// TwinCAT 3 PLC project pruebaAlmacenje
// ProgramVersion: 3.1.4024.0
// libraries:
//   Tc2_Standard, * (Beckhoff Automation GmbH)
//   Tc2_System, * (Beckhoff Automation GmbH)
//   Tc3_Module, * (Beckhoff Automation GmbH)
//   VisuSymbols,3.5.10.0,System
// project tree:
//   / GlobalTextList.TcGTLO, PlcTask.TcTTO (not stored), Visualization Manager.TcVMO (not stored)
//   GVLs/ GVLvar.TcGVL
//   POUs/ inicializarPosOcupEstanteria.TcPOU, MAIN.TcPOU, posicionEstanteria.TcPOU, distanciaBaldas.TcPOU
//   VISUs/ equivalenciaBaldaOcupada.TcTLO, HMI.TcVIS
// real-time tasks:
//   TASK PlcTask: cycle T#10ms, priority 20, ADS port 350

// ---- GVLs/GVLvar.TcGVL
{attribute 'qualified_only'}
VAR_GLOBAL
	
	// Cuadro
	{attribute 'OPC.UA.DA' := '1'}
	botonStart : BOOL;
	{attribute 'OPC.UA.DA' := '1'}
	botonStop : BOOL;
	{attribute 'OPC.UA.DA' := '1'}
	botonReset : BOOL; 
	{attribute 'OPC.UA.DA' := '1'}
	seta: BOOL;
	{attribute 'OPC.UA.DA' := '1'}
	luzVerde : BOOL;
	{attribute 'OPC.UA.DA' := '1'}
	luzAmarillo : BOOL;
	{attribute 'OPC.UA.DA' := '1'}
	luzRoja : BOOL;
	{attribute 'OPC.UA.DA' := '1'}
	luzBotonStart : BOOL;
	{attribute 'OPC.UA.DA' := '1'}
	luzBotonStop :  BOOL;
	{attribute 'OPC.UA.DA' := '1'}
	luzBotonReset : BOOL;
	{attribute 'OPC.UA.DA' := '1'}
	modoManual : BOOL;
	{attribute 'OPC.UA.DA' := '1'}
	modoAuto : BOOL;
	
	

	// Estanterias
	estanteria: ARRAY[1..6,1..6] OF ARRAY[1..2] OF REAL;
	baldasOcupadas : ARRAY [1..6,1..3] OF BOOL;
	
	// Cintas
	{attribute 'OPC.UA.DA' := '1'}
	cinta : BOOL;
	{attribute 'OPC.UA.DA' := '1'}
	cintaTransportadoraPalet : BOOL; 

	// Grua
	{attribute 'OPC.UA.DA' := '1'}
	moveForksLeft : BOOL; // horquilla hacia ixquierda
	{attribute 'OPC.UA.DA' := '1'}
	moveForksRight : BOOL; // hoquilla hacia derecha
	//{attribute 'OPC.UA.DA' := '1'}
	//elevacionLigeraPlataforma : BOOL;
	{attribute 'OPC.UA.DA' := '1'}
	movingZ : REAL; // actual poscion en Z
	{attribute 'OPC.UA.DA' := '1'}
	movingX : REAL; // actual posicion en X
	{attribute 'OPC.UA.DA' := '1'}
	forkLeftLimit : BOOL; 
	{attribute 'OPC.UA.DA' := '1'}
	forkMiddleLimit : BOOL;
	{attribute 'OPC.UA.DA' := '1'}
	forkRightLimit : BOOL;
	{attribute 'OPC.UA.DA' := '1'}
	setPointX : REAL; // movimientp columnas (horizontal)
	{attribute 'OPC.UA.DA' := '1'}
	setPointZ : REAL; // movimeinto filas (vertical)
	
	//sensores
	{attribute 'OPC.UA.DA' := '1'}
	sensorEntradaGrua : bool;


END_VAR

// ---- POUs/inicializarPosOcupEstanteria.TcPOU
FUNCTION_BLOCK inicializarPosOcupEstanteria
VAR_INPUT
END_VAR
VAR_OUTPUT
END_VAR
VAR
	i: INT;
	fila: INT;
	col: INT;
END_VAR

// Se inicializan las posicones del amlmcen a false
// por defecto se empieza con el almacen vacio
FOR fila := 1 TO 6 DO
    FOR col := 1 TO 3 DO
        // la primera posicion libre 
		 GVLvar.baldasOcupadas[fila,col] := FALSE;
    END_FOR
END_FOR

END_FUNCTION_BLOCK

// ---- POUs/MAIN.TcPOU
PROGRAM MAIN
VAR
	enclaveStart: BOOL;
	timerColumna: TON;
	posicionEst : ARRAY[1..4] OF REAL;
	distBaldas : distanciaBaldas();
	iniPosOcupEst : inicializarPosOcupEstanteria();
	cargando: BOOL;
	flancoMovingX : F_TRIG;
	flancoMovingZ : F_TRIG;
	movingZ: BOOL;
	movingX: BOOL;
	descragandoElem: BOOL;
	descargandoElem: BOOL;
	elemDescargado: BOOL;
	state: INT := 1;
	posInicialZ : real := 0.2;
	horquillaExtendida: BOOL;
	timerExternsionHorquilla: TON;
	startTimerHorquilla: BOOL;
	timerExtension: BOOL;
	posActual: REAL;
	bajarHorquilla: BOOL;
	timerBajarHorquilla: TON;
	incfementoBaizadaH : REAL := 0.4;
	enPosicoin: BOOL;
	posmovingZ: REAL;
	luzStart :bool;
	luzReset: BOOL;
	luzStop : bool;
	luzVerde: BOOL;
	luzAmarilla: BOOL;
	luzRoja: BOOL;
	emergencia: BOOL;
	cinta:bool;
	setPointX: REAL;
	setPointZ: REAL;
	cintaTransportadoraPalet: BOOL;
	botonReset: BOOL;
	seta : bool;
	botonStart: BOOL;
	botonStop: BOOL;
	filaEstanteria: INT;
	colEstanteria: INT;
	moving: REAL;
END_VAR

VAR PERSISTENT
	elemCargado: BOOL;
END_VAR

// ----------------------------- Logica Botones ----------------------------------------

//Luces Botons
luzStart := FALSE;
luzStop := FALSE;
luzReset:=FALSE;

(*Boton start 



*)
IF GVLvar.botonStart AND NOT emergencia THEN
	luzStart:= TRUE;
	luzVerde := TRUE;
	luzAmarilla := FALSE;
	luzRoja := FALSE;
	enclaveStart := TRUE;
	cinta := TRUE;
	cintaTransportadoraPalet := TRUE; 
	distBaldas();
	iniPosOcupEst();
	setPointZ := 0.2;
END_IF

IF NOT GVLvar.botonStop AND NOT emergencia THEN
	luzStop := TRUE;
	luzVerde := FALSE;
	luzAmarilla := TRUE;
	luzRoja := FALSE;
	enclaveStart := FALSE;
	cinta := FALSE;
	cintaTransportadoraPalet := FALSE;
END_IF


IF  NOT GVLvar.seta THEN
	luzRoja:= TRUE;
	luzVerde := FALSE;
	luzAmarilla := FALSE;
	
	emergencia := TRUE;
	cinta := FALSE;
	cintaTransportadoraPalet := FALSE	; 
	enclaveStart := FALSE;
END_IF


IF  GVLvar.seta AND emergencia THEN
	IF GVLvar.botonReset THEN
		emergencia := FALSE;
		cinta := TRUE;
		cintaTransportadoraPalet := TRUE; 
		enclaveStart := TRUE;
		luzRoja := FALSE;
		luzVerde := TRUE;
		luzAmarilla := FALSE;
	END_IF	
END_IF

// ---------------------------------------------------------------------

IF enclaveStart THEN
	

	CASE state OF
	
		// 1. Esperando Start
		1: 
//			IF GVLvar.botonStart THEN
//				enclaveStart := TRUE;
//				GVLvar.cinta := TRUE;
//				distBaldas();
//				iniPosOcupEst();
//				GVLvar.setPointZ := 0.3;
//				state := 2;  // pasar al siguiente estado
//			END_IF
			setPointZ := posInicialZ;
			state := 2;  // pasar al siguiente estado
			
		// 2. Espera caja en la entrada
		2:
			IF GVLvar.sensorEntradaGrua THEN
				cinta := FALSE;
				cintaTransportadoraPalet := FALSE;
				GVLvar.moveForksRight := TRUE;
				state := 3;
			END_IF
	
		// 3. Horquilla desplegando
		3:
			IF GVLvar.forkRightLimit THEN
				setPointZ := posInicialZ + 0.2;
				startTimerHorquilla := TRUE;
			END_IF
			
			timerExternsionHorquilla (IN:=startTimerHorquilla, PT:= T#2S);
			
			horquillaExtendida :=  (GVLvar.movingZ = (posInicialZ + 0.2)) OR (GVLvar.movingZ > ((posInicialZ + 0.2)-0.05)) OR (GVLvar.movingZ < ((posInicialZ + 0.2)+0.05));
			//IF GVLvar.movingZ = (posInicialZ + 0.2) THEN
			IF timerExternsionHorquilla.Q AND horquillaExtendida THEN
				GVLvar.moveForksRight := FALSE;
				elemCargado := TRUE;
				startTimerHorquilla := FALSE;
				state := 4;
			END_IF
			
//			IF GVLvar.forkMiddleLimit  AND elemCargado THEN 
				
				
//			END_IF
	
		// 4. Calcular posición libre y mover X/Z
		4:
			IF elemCargado AND GVLvar.forkMiddleLimit THEN 
				posicionEst := posicionEstanteria();
				// Si devuelve una posicion valida
				IF posicionEst[1]<>0 AND posicionEst[2]<>0 THEN
					setPointX := posicionEst[1];   // columna (X)
					setPointZ := posicionEst[2]+0.4;   // fila (Z)
					filaEstanteria := TO_INT(posicionEst[3]);
					colEstanteria := TO_INT(posicionEst[4]);
					elemCargado := FALSE;
					descargandoElem := TRUE;
					state := 5;
				END_IF
			END_IF
	
		// 5. Esperar llegar a destino
		5:
			 movingX := (GVLvar.movingX = posicionEst[1]) OR (GVLvar.movingX > (posicionEst[1]-0.05) AND GVLvar.movingX < posicionEst[1]) OR (GVLvar.movingX < (posicionEst[1]+0.05)AND GVLvar.movingX > posicionEst[1]) ;
			 movingZ := (GVLvar.movingZ = posicionEst[2]+0.4) OR (GVLvar.movingZ > (posicionEst[2]-0.05+0.4) AND GVLvar.movingZ < posicionEst[2]+0.4) OR (GVLvar.movingZ < (posicionEst[2]+0.05+0.4) AND GVLvar.movingZ > posicionEst[2]+0.4);
			 
			 
			IF movingZ AND movingX AND descargandoElem THEN
				GVLvar.moveForksLeft := TRUE;
				bajarHorquilla := TRUE;
				state := 6;
			END_IF
			
			
		6:	
			//timerBajarHorquilla (IN:= bajarHorquilla, PT:=T#2S);
			
			//IF  enPosicoin AND GVLvar.forkMiddleLimit THEN  
			IF GVLvar.forkLeftLimit THEN
				 moving := GVLvar.movingZ;
				IF moving > 0 THEN 
					setPointZ := GVLvar.movingZ - incfementoBaizadaH ;	
				END_IF
				descargandoElem := FALSE;
				bajarHorquilla := FALSE;
				state := 7;
			END_IF
			
		// 6. Horquilla descargando
		7:
			posmovingZ := GVLvar.movingZ;	
			enPosicoin  := (posmovingZ = posicionEst[2]) OR (posmovingZ > (posicionEst[2] -0.05) AND posmovingZ < posicionEst[2]) OR (posmovingZ < (posicionEst[2]+0.05) AND posmovingZ > posicionEst[2]);
			 
			IF GVLvar.forkLeftLimit AND enPosicoin THEN
				GVLvar.moveForksLeft := FALSE;
				elemDescargado := TRUE;
				state := 8;
       		END_IF
			
		
			
		// 7. Volver a origen
		8:
			IF elemDescargado AND GVLvar.forkMiddleLimit THEN
				setPointX := 0.0;
				setPointZ :=posInicialZ;
				elemDescargado := FALSE;
				cinta := TRUE;
				cintaTransportadoraPalet := TRUE; 
				state := 2;
			END_IF
	
	//    // 8. Reanudar cinta y volver a esperar
	//    8:
	//        IF (GVLvar.movingX = 0.0) AND (GVLvar.movingZ = 0.3) THEN
	//            GVLvar.cinta := TRUE;
	//            state := 2;   // vuelve a esperar siguiente caja
	//        END_IF
	
		// Estado por defecto (seguridad)
		ELSE
			state := 1;
	
	END_CASE
END_IF


// ----------------------------- Actualizar Salidas  ----------------------------------------
GVLvar.setPointX := setPointX;
GVLvar.setPointZ := setPointZ;

GVLvar.luzAmarillo := luzAmarilla;
GVLvar.luzVerde := luzVerde;
GVLvar.luzRoja := luzRoja;
GVLvar.luzBotonReset := luzReset;
GVLvar.luzBotonStart := luzStart;
GVLvar.luzBotonStop := luzStop;

GVLvar.cinta := cinta;
GVLvar.cintaTransportadoraPalet := cintaTransportadoraPalet;


//GVLvar.seta := seta;
//GVLvar.botonReset := botonReset;
//GVLvar.botonStart := botonStart;
//GVLvar.botonStop := botonStop:

END_PROGRAM

// ---- POUs/distanciaBaldas.TcPOU
FUNCTION_BLOCK distanciaBaldas
VAR_INPUT
END_VAR
VAR_OUTPUT
END_VAR
VAR
END_VAR

// Fila 1
GVLvar.estanteria[1,1][1] := 1.55;  GVLvar.estanteria[1,1][2] := 0.5;
GVLvar.estanteria[1,2][1] := 2.6;  GVLvar.estanteria[1,2][2] := 0.5;
GVLvar.estanteria[1,3][1] := 3.7;  GVLvar.estanteria[1,3][2] := 0.5;

// Fila 2
GVLvar.estanteria[2,1][1] := 1.55;  GVLvar.estanteria[2,1][2] := 2.1;
GVLvar.estanteria[2,2][1] := 2.6;  GVLvar.estanteria[2,2][2] := 2.1;
GVLvar.estanteria[2,3][1] := 3.7;  GVLvar.estanteria[2,3][2] := 2.1;

// Fila 3
GVLvar.estanteria[3,1][1] := 1.65;  GVLvar.estanteria[3,1][2] := 3.9;
GVLvar.estanteria[3,2][1] := 2.6;  GVLvar.estanteria[3,2][2] := 3.9;
GVLvar.estanteria[3,3][1] := 3.7;  GVLvar.estanteria[3,3][2] := 3.9;

// Fila 4
GVLvar.estanteria[4,1][1] := 1.6;  GVLvar.estanteria[4,1][2] := 5.6;
GVLvar.estanteria[4,2][1] := 2.6;  GVLvar.estanteria[4,2][2] := 5.6;
GVLvar.estanteria[4,3][1] := 3.7;  GVLvar.estanteria[4,3][2] := 5.6;

// Fila 5
GVLvar.estanteria[5,1][1] := 1.6;  GVLvar.estanteria[5,1][2] := 8.3;
GVLvar.estanteria[5,2][1] := 2.6;  GVLvar.estanteria[5,2][2] := 8.3;
GVLvar.estanteria[5,3][1] := 3.7;  GVLvar.estanteria[5,3][2] := 8.3;

// Fila 6
GVLvar.estanteria[6,1][1] := 1.6;  GVLvar.estanteria[6,1][2] := 8.7;
GVLvar.estanteria[6,2][1] := 2.6;  GVLvar.estanteria[6,2][2] := 8.7;
GVLvar.estanteria[6,3][1] := 3.7;  GVLvar.estanteria[6,3][2] := 8.7;

END_FUNCTION_BLOCK

// ---- POUs/posicionEstanteria.TcPOU
FUNCTION posicionEstanteria : Array[1..4] of real
VAR_INPUT
END_VAR
VAR
	posicion : ARRAY[1..2] OF REAL;
	// 1 - posicion en X (horizontal)
	// 2 - posicoin en Z (vertical)
	fila: DINT;
	arr2D: INT;
	col: DINT;
	encontrado: BOOL;
END_VAR

encontrado  := FALSE;
FOR fila := 1 TO 6 DO
    FOR col := 1 TO 3 DO
        // la primera posicion libre 
		IF GVLvar.baldasOcupadas[fila,col] = FALSE  AND encontrado = FALSE THEN
			posicionEstanteria[1] := GVLvar.estanteria[fila,col][1];
			posicionEstanteria[2] := GVLvar.estanteria[fila,col][2];
			posicionEstanteria[3] := TO_REAL(fila) ;
			posicionEstanteria[4] := TO_REAL(col);
			
			GVLvar.baldasOcupadas[fila,col] := TRUE;
			encontrado := TRUE;
			EXIT;
//		ELSE 
//			posicionEstanteria := [0,0];
		END_IF
    END_FOR
END_FOR

END_FUNCTION

// ---- GlobalTextList.TcGTLO
TEXTLIST GlobalTextList
  538 = '%B'
  557 = '%b'
  838 = '%i'
  837 = 'Cargando Palet'
  351 = 'Descargando Palet'
  912 = 'ESTANTERÍA'
  378 = 'FiColumnala'
  976 = 'Fila'
  655 = 'GRÚA'
  699 = 'GRÚA DESPLAZANDOSE A'
  528 = 'Horquilla en reposo'
  343 = 'Horquilla extendida Dcha'
  803 = 'Horquilla extendida Izq'
  777 = 'Indicador de mesa giratoria orientada a 90º'
  953 = 'Indicador de mesa giratoria orinetada a 0ª (posicion de reposo)'
  894 = 'Indicador de un palet sobre la mesa giratoria'
  359 = 'Mesa en 0º'
  512 = 'Mesa en 90º'
  134 = 'MESA GIRATORIA'
  194 = 'Palet en Mesa'
  465 = 'Posicion'
  379 = 'Posición '
  139 = 'Reset'
  163 = 'Seta'
  56 = 'Seta Emergencia'
  759 = 'Start'
  420 = 'Stop'
END_TEXTLIST

// ---- VISUs/equivalenciaBaldaOcupada.TcTLO
TEXTLIST equivalenciaBaldaOcupada
  TRUE = 'Ocupada'
  FALSE = 'Libre'
   = ''
END_TEXTLIST

// ---- VISUs/HMI.TcVIS
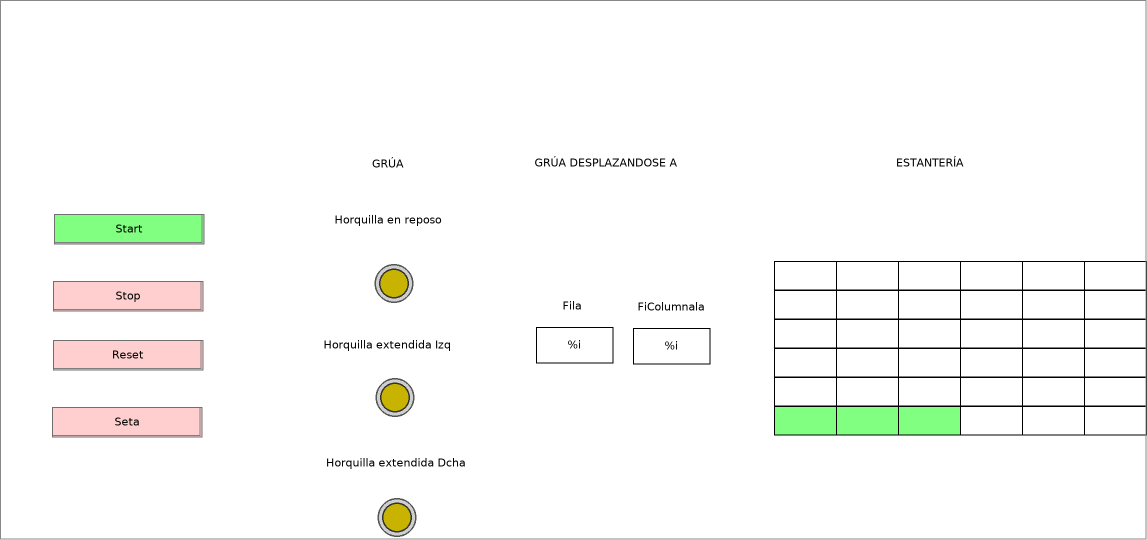
VISUALIZATION HMI  // 1147x540
    Button (54,214 150x30), "Start"
        toggle GVLvar.botonStart
    Button (53,281 150x30), "Stop", colour toggle: NOT GVLvars.botonStop
        toggle GVLvar.botonStop
    Button (53,340 150x30), "Reset", colour toggle: GVLvars.botonReset
        toggle GVLvar.botonReset
    Button (52,407 150x30), "Seta", colour toggle: GVLvars.seta
        toggle not GVLvars.seta
    Lamp1 (368,261 52x45), tooltip "Indicador de un palet sobre la mesa giratoria", variable: GVLvars.frontLimit, style: Lamp-Lamp1-Yellow
    Label (313,149 150x30), "GRÚA"
    Lamp1 (369,375 52x45), tooltip "Indicador de mesa giratoria orientada a 90º", variable: GVLvars.maximunRotation, style: Lamp-Lamp1-Yellow
    Label (308,330 159x30), "Horquilla extendida Izq"
    Label (313,205 150x30), "Horquilla en reposo"
    Lamp1 (371,495 52x45), tooltip "Indicador de mesa giratoria orinetada a 0ª (posicion de reposo)", variable: GVLvars.minuminRotation, style: Lamp-Lamp1-Yellow
    Label (322,448 148x30), "Horquilla extendida Dcha"
    Rectangle (536,327 77x36), "%i", text variable: MAIN.filaEstanteria
    Label (557,291 30x30), "Fila"
    Rectangle (633,328 77x36), "%i", text variable: MAIN.colEstanteria
    Label (645,292 52x30), "FiColumnala"
    RoundedRectangle (774,261 63x29)
    RoundedRectangle (836,261 63x29)
    RoundedRectangle (898,261 63x29)
    RoundedRectangle (960,261 63x29)
    RoundedRectangle (1022,261 63x29)
    RoundedRectangle (1084,261 63x29)
    RoundedRectangle (774,290 63x29)
    RoundedRectangle (836,290 63x29)
    RoundedRectangle (898,290 63x29)
    RoundedRectangle (960,290 63x29)
    RoundedRectangle (1022,290 63x29)
    RoundedRectangle (1084,290 63x29)
    RoundedRectangle (774,319 63x29)
    RoundedRectangle (836,319 63x29)
    RoundedRectangle (898,319 63x29)
    RoundedRectangle (960,319 63x29)
    RoundedRectangle (1022,319 63x29)
    RoundedRectangle (1084,319 63x29)
    RoundedRectangle (774,348 63x29)
    RoundedRectangle (836,348 63x29)
    RoundedRectangle (898,348 63x29)
    RoundedRectangle (960,348 63x29)
    RoundedRectangle (1022,348 63x29)
    RoundedRectangle (1084,348 63x29)
    RoundedRectangle (774,377 63x29)
    RoundedRectangle (836,377 63x29)
    RoundedRectangle (898,377 63x29)
    RoundedRectangle (960,377 63x29)
    RoundedRectangle (1022,377 63x29)
    RoundedRectangle (1084,377 63x29)
    RoundedRectangle (774,406 63x29), text list: 'equivalenciaBaldaOcupada', text index: GVLvar.baldasOcupadas[1][1]
        p2167032090: not GVLvar.baldasOcupadas[1][1]
        p3092690914: GVLvar.baldasOcupadas[1][1]
    RoundedRectangle (836,406 63x29), colour toggle: GVLvar.baldasOcupadas[1][2]
    RoundedRectangle (898,406 63x29), colour toggle: GVLvar.baldasOcupadas[1][3]
    RoundedRectangle (960,406 63x29)
    RoundedRectangle (1022,406 63x29)
    RoundedRectangle (1084,406 63x29)
    Label (515,148 182x30), "GRÚA DESPLAZANDOSE A"
    Label (855,148 150x30), "ESTANTERÍA"
END_VISUALIZATION
